{attribute 'qualified_only'}
VAR_GLOBAL RETAIN
		Value :INT:=2;
END_VAR

(* stored: Version 1.1.0.1, ProductVersion 3.1.4024.4
   GVL GLV_USER_FUN: Id {10e41103-96e0-4120-ab4a-46571acc69a8} *)
